// TIA Portal V20 export
FUNCTION "CALL_OPMODE_PANEL_FC" : Void   // FC200, LAD
TITLE = Aufruf Pult / Betriebsart / Call panels / operating modes
{ S7_Optimized_Access := 'TRUE' }
FAMILY : Base
VERSION : 1.0
// FUNKTIONSBESCHREIBUNG:
// Der Baustein dient als Aufrufschnittstelle für die HMI-/Panel- und Betriebsartenbausteine.
// Weitere Hinweise: siehe SICAR anwenderdefinierte Dokumentation / SICAR Online-Hilfe.
// DESCRIPTION OF FUNCTIONS:
// This function is the calling interface for initialization HMI/Panel and Operation mode blocks.
// For more informations see Tesla userdefined documentation / online-help.
// 描述 OF 功能:
// 这个 功能 is  calling 接口 给 初始化 HMI/Panel 和 运行 模式 blocks.
// 给 more informations see SICAR userdefined documentation / SICAR online-帮助.
// stored: AutoNumber false, SetENOAutomatically false
   VAR_TEMP
      Auxiliary_flag : Bool;
      Dummy_byte : Byte;
      dummy_word : Word;
      ParaAlarm : USInt;
      "020RB01_SlowDown" : Bool;
      "020RB02_SlowDown" : Bool;
      "020RB03_SlowDown" : Bool;
      "020RB04_SlowDown" : Bool;
      "020RB06_SlowDown" : Bool;
      "025RB01_SlowDown" : Bool;
      "025RB02_SlowDown" : Bool;
      "030RB01_SlowDown" : Bool;
      "030RB02_SlowDown" : Bool;
      "030RB03_SlowDown" : Bool;
      "030RB04_SlowDown" : Bool;
      待关联外部按钮1 : Bool;
      待关联外部按钮2 : Bool;
      待关联外部按钮2_1 : Bool;
   END_VAR
   VAR_TEMP   // added for the SCL form of the ladder/FBD networks
      _w1 : Bool;
      _w2 : Bool;
   END_VAR
BEGIN

REGION Network 1: Aufruf: HMI 1 / Call Operatorpanel_01: UBM1+010-HMI02 / Call: HMI_1
   // 介绍：设置和管理操作面板，
   // HMI:控制操作模式，可视化屏幕，
   // Panel：控制操作模式，按钮盒，
   // 有几个HMI调用几次，每次调用都需要对其定义类型。
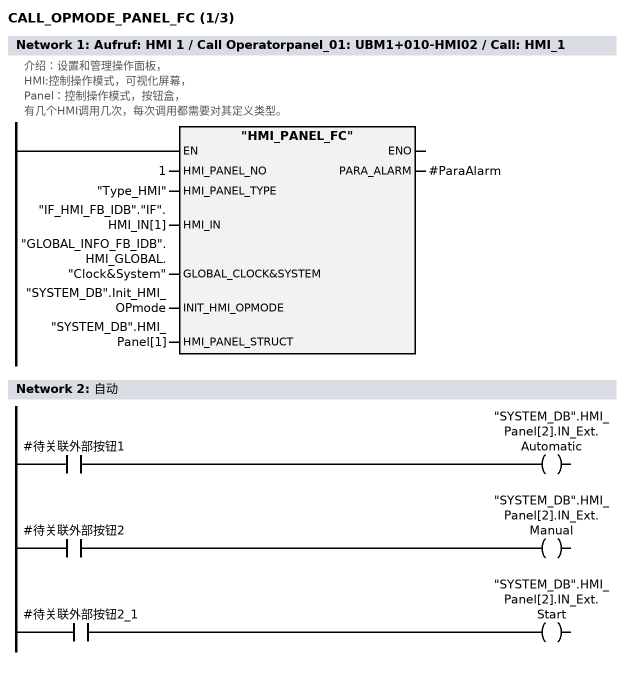
   RUNG wire#powerrail
      "HMI_PANEL_FC"(HMI_PANEL_NO := 1, HMI_PANEL_TYPE := "Type_HMI", HMI_IN := "IF_HMI_FB_IDB"."IF".HMI_IN[1], "GLOBAL_CLOCK&SYSTEM" := "GLOBAL_INFO_FB_IDB".HMI_GLOBAL."Clock&System", INIT_HMI_OPMODE := "SYSTEM_DB".Init_HMI_OPmode, HMI_PANEL_STRUCT := "SYSTEM_DB".HMI_Panel[1], PARA_ALARM => #ParaAlarm)
   END_RUNG
   // the same network as SCL:
   "HMI_PANEL_FC"(HMI_PANEL_NO := 1,
                  HMI_PANEL_TYPE := "Type_HMI",
                  HMI_IN := "IF_HMI_FB_IDB"."IF".HMI_IN[1],
                  "GLOBAL_CLOCK&SYSTEM" := "GLOBAL_INFO_FB_IDB".HMI_GLOBAL."Clock&System",
                  INIT_HMI_OPMODE := "SYSTEM_DB".Init_HMI_OPmode,
                  HMI_PANEL_STRUCT := "SYSTEM_DB".HMI_Panel[1],
                  PARA_ALARM => #ParaAlarm);
END_REGION

REGION Network 2: 自动
   RUNG wire#powerrail
      Contact( #待关联外部按钮1 )
      Coil( "SYSTEM_DB".HMI_Panel[2].IN_Ext.Automatic )
   END_RUNG
   RUNG wire#powerrail
      Contact( #待关联外部按钮2 )
      Coil( "SYSTEM_DB".HMI_Panel[2].IN_Ext.Manual )
   END_RUNG
   RUNG wire#powerrail
      Contact( #待关联外部按钮2_1 )
      Coil( "SYSTEM_DB".HMI_Panel[2].IN_Ext.Start )
   END_RUNG
   // the same network as SCL:
   "SYSTEM_DB".HMI_Panel[2].IN_Ext.Automatic := #待关联外部按钮1;
   "SYSTEM_DB".HMI_Panel[2].IN_Ext.Manual := #待关联外部按钮2;
   "SYSTEM_DB".HMI_Panel[2].IN_Ext.Start := #待关联外部按钮2_1;
END_REGION

REGION Network 3: E-Stop / Call: 运行 模式 area 1 - Create 新的 OpMode
   // 介绍：设置和管理操作操作模式OPMode，有几个OPMode就需要调用几次，每次调用都需要对其与HMI的关系进行定义。
   // 一个OPMode至少需要一个HMI/pannei控制；
   // 一个HMI/Panel可以控制多个OPMode；
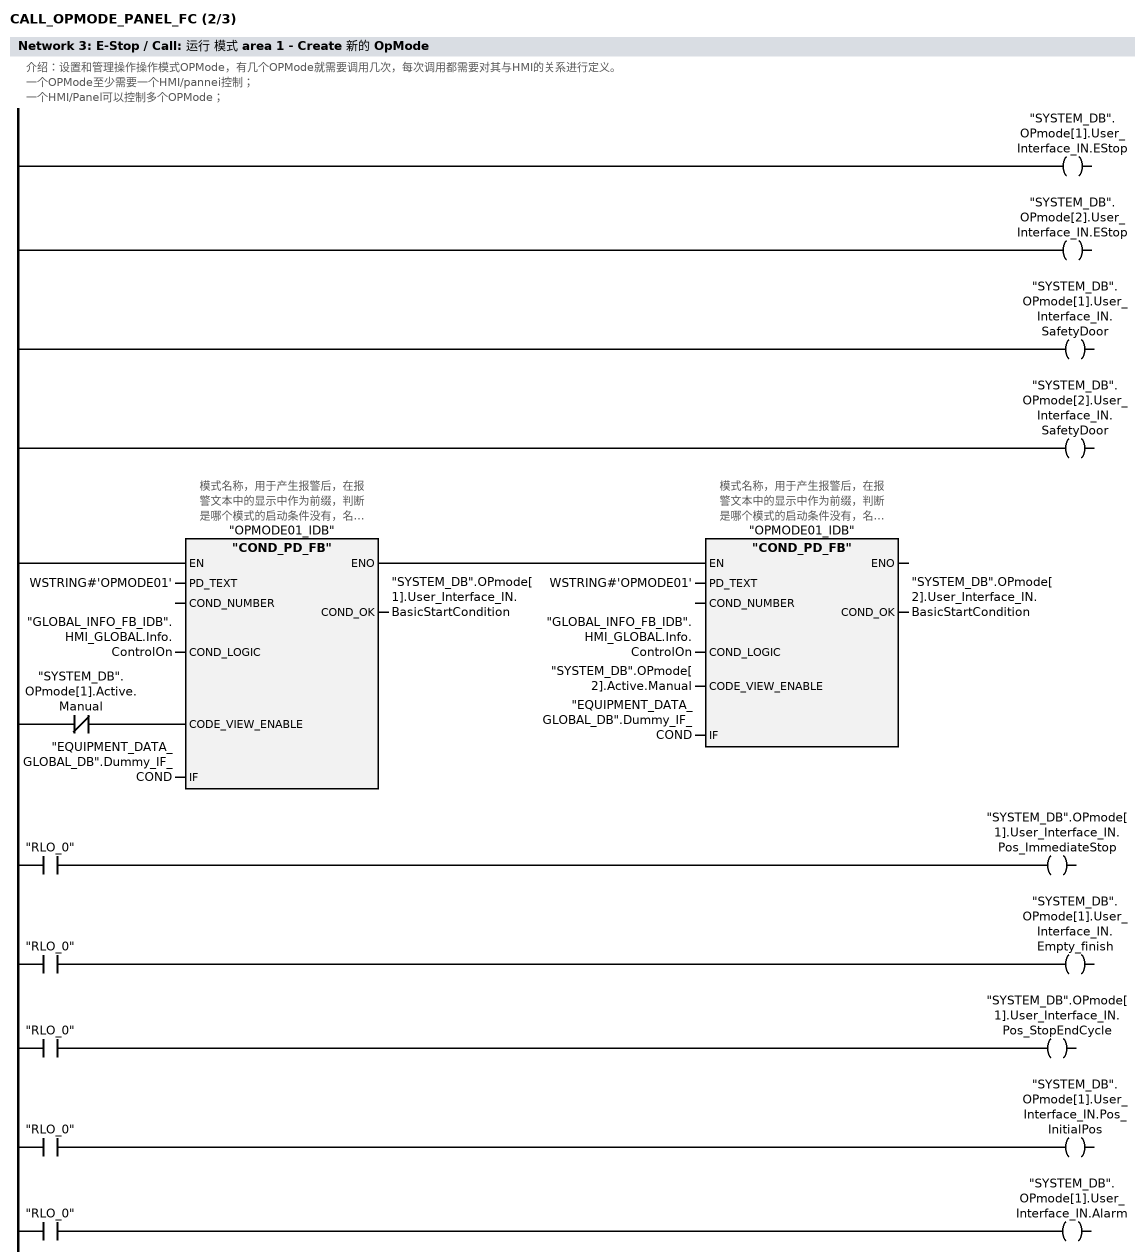
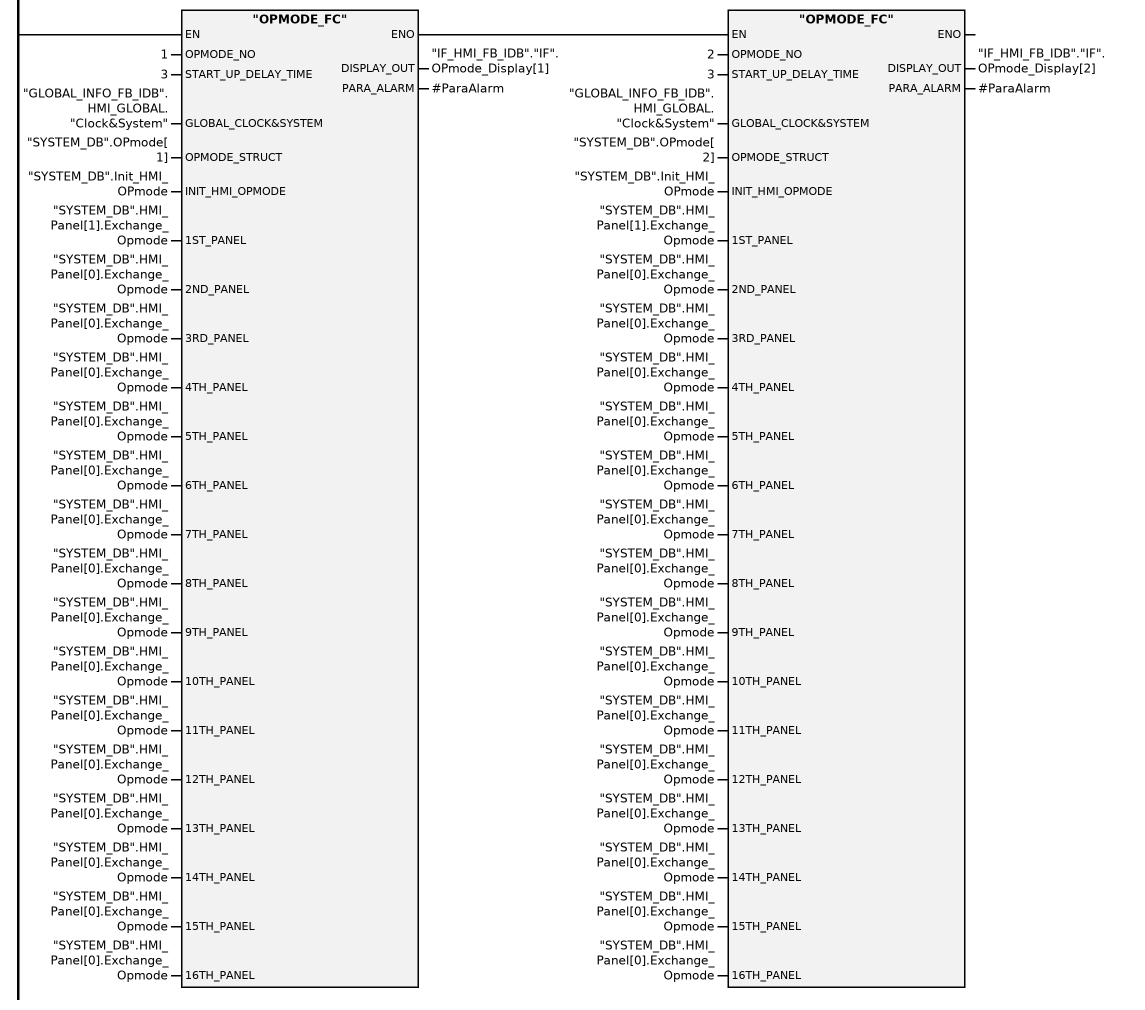
   RUNG wire#powerrail
      Coil( "SYSTEM_DB".OPmode[1].User_Interface_IN.EStop )
   END_RUNG
   RUNG wire#powerrail
      Coil( "SYSTEM_DB".OPmode[2].User_Interface_IN.EStop )
   END_RUNG
   RUNG wire#powerrail
      Coil( "SYSTEM_DB".OPmode[1].User_Interface_IN.SafetyDoor )
   END_RUNG
   RUNG wire#powerrail
      Coil( "SYSTEM_DB".OPmode[2].User_Interface_IN.SafetyDoor )
   END_RUNG
   RUNG wire#powerrail
      "OPMODE01_IDB"(CODE_VIEW_ENABLE := wire#w1, PD_TEXT := WSTRING#'OPMODE01', COND_NUMBER :=, COND_LOGIC := "GLOBAL_INFO_FB_IDB".HMI_GLOBAL.Info.ControlOn, "IF" := "EQUIPMENT_DATA_GLOBAL_DB".Dummy_IF_COND, COND_OK => "SYSTEM_DB".OPmode[1].User_Interface_IN.BasicStartCondition)   // 模式名称，用于产生报警后，在报警文本中的显示中作为前缀，判断是哪个模式的启动条件没有，名称已经预先填写在了对应DB块数据中
      "OPMODE01_IDB"(PD_TEXT := WSTRING#'OPMODE01', COND_NUMBER :=, COND_LOGIC := "GLOBAL_INFO_FB_IDB".HMI_GLOBAL.Info.ControlOn, CODE_VIEW_ENABLE := "SYSTEM_DB".OPmode[2].Active.Manual, "IF" := "EQUIPMENT_DATA_GLOBAL_DB".Dummy_IF_COND, COND_OK => "SYSTEM_DB".OPmode[2].User_Interface_IN.BasicStartCondition)   // 模式名称，用于产生报警后，在报警文本中的显示中作为前缀，判断是哪个模式的启动条件没有，名称已经预先填写在了对应DB块数据中
   END_RUNG
   RUNG wire#powerrail
      I_Contact( "SYSTEM_DB".OPmode[1].Active.Manual )
   END_RUNG wire#w1
   RUNG wire#powerrail
      Contact( "RLO_0" )
      Coil( "SYSTEM_DB".OPmode[1].User_Interface_IN.Pos_ImmediateStop )
   END_RUNG
   RUNG wire#powerrail
      Contact( "RLO_0" )
      Coil( "SYSTEM_DB".OPmode[1].User_Interface_IN.Empty_finish )
   END_RUNG
   RUNG wire#powerrail
      Contact( "RLO_0" )
      Coil( "SYSTEM_DB".OPmode[1].User_Interface_IN.Pos_StopEndCycle )
   END_RUNG
   RUNG wire#powerrail
      Contact( "RLO_0" )
      Coil( "SYSTEM_DB".OPmode[1].User_Interface_IN.Pos_InitialPos )
   END_RUNG
   RUNG wire#powerrail
      Contact( "RLO_0" )
      Coil( "SYSTEM_DB".OPmode[1].User_Interface_IN.Alarm )
   END_RUNG
   RUNG wire#powerrail
      "OPMODE_FC"(OPMODE_NO := 1, START_UP_DELAY_TIME := 3, "GLOBAL_CLOCK&SYSTEM" := "GLOBAL_INFO_FB_IDB".HMI_GLOBAL."Clock&System", OPMODE_STRUCT := "SYSTEM_DB".OPmode[1], INIT_HMI_OPMODE := "SYSTEM_DB".Init_HMI_OPmode, "1ST_PANEL" := "SYSTEM_DB".HMI_Panel[1].Exchange_Opmode, "2ND_PANEL" := "SYSTEM_DB".HMI_Panel[0].Exchange_Opmode, "3RD_PANEL" := "SYSTEM_DB".HMI_Panel[0].Exchange_Opmode, "4TH_PANEL" := "SYSTEM_DB".HMI_Panel[0].Exchange_Opmode, "5TH_PANEL" := "SYSTEM_DB".HMI_Panel[0].Exchange_Opmode, "6TH_PANEL" := "SYSTEM_DB".HMI_Panel[0].Exchange_Opmode, "7TH_PANEL" := "SYSTEM_DB".HMI_Panel[0].Exchange_Opmode, "8TH_PANEL" := "SYSTEM_DB".HMI_Panel[0].Exchange_Opmode, "9TH_PANEL" := "SYSTEM_DB".HMI_Panel[0].Exchange_Opmode, "10TH_PANEL" := "SYSTEM_DB".HMI_Panel[0].Exchange_Opmode, "11TH_PANEL" := "SYSTEM_DB".HMI_Panel[0].Exchange_Opmode, "12TH_PANEL" := "SYSTEM_DB".HMI_Panel[0].Exchange_Opmode, "13TH_PANEL" := "SYSTEM_DB".HMI_Panel[0].Exchange_Opmode, "14TH_PANEL" := "SYSTEM_DB".HMI_Panel[0].Exchange_Opmode, "15TH_PANEL" := "SYSTEM_DB".HMI_Panel[0].Exchange_Opmode, "16TH_PANEL" := "SYSTEM_DB".HMI_Panel[0].Exchange_Opmode, DISPLAY_OUT => "IF_HMI_FB_IDB"."IF".OPmode_Display[1], PARA_ALARM => #ParaAlarm)
      "OPMODE_FC"(OPMODE_NO := 2, START_UP_DELAY_TIME := 3, "GLOBAL_CLOCK&SYSTEM" := "GLOBAL_INFO_FB_IDB".HMI_GLOBAL."Clock&System", OPMODE_STRUCT := "SYSTEM_DB".OPmode[2], INIT_HMI_OPMODE := "SYSTEM_DB".Init_HMI_OPmode, "1ST_PANEL" := "SYSTEM_DB".HMI_Panel[1].Exchange_Opmode, "2ND_PANEL" := "SYSTEM_DB".HMI_Panel[0].Exchange_Opmode, "3RD_PANEL" := "SYSTEM_DB".HMI_Panel[0].Exchange_Opmode, "4TH_PANEL" := "SYSTEM_DB".HMI_Panel[0].Exchange_Opmode, "5TH_PANEL" := "SYSTEM_DB".HMI_Panel[0].Exchange_Opmode, "6TH_PANEL" := "SYSTEM_DB".HMI_Panel[0].Exchange_Opmode, "7TH_PANEL" := "SYSTEM_DB".HMI_Panel[0].Exchange_Opmode, "8TH_PANEL" := "SYSTEM_DB".HMI_Panel[0].Exchange_Opmode, "9TH_PANEL" := "SYSTEM_DB".HMI_Panel[0].Exchange_Opmode, "10TH_PANEL" := "SYSTEM_DB".HMI_Panel[0].Exchange_Opmode, "11TH_PANEL" := "SYSTEM_DB".HMI_Panel[0].Exchange_Opmode, "12TH_PANEL" := "SYSTEM_DB".HMI_Panel[0].Exchange_Opmode, "13TH_PANEL" := "SYSTEM_DB".HMI_Panel[0].Exchange_Opmode, "14TH_PANEL" := "SYSTEM_DB".HMI_Panel[0].Exchange_Opmode, "15TH_PANEL" := "SYSTEM_DB".HMI_Panel[0].Exchange_Opmode, "16TH_PANEL" := "SYSTEM_DB".HMI_Panel[0].Exchange_Opmode, DISPLAY_OUT => "IF_HMI_FB_IDB"."IF".OPmode_Display[2], PARA_ALARM => #ParaAlarm)
   END_RUNG
   // the same network as SCL:
   "SYSTEM_DB".OPmode[1].User_Interface_IN.EStop := TRUE;
   "SYSTEM_DB".OPmode[2].User_Interface_IN.EStop := TRUE;
   "SYSTEM_DB".OPmode[1].User_Interface_IN.SafetyDoor := TRUE;
   "SYSTEM_DB".OPmode[2].User_Interface_IN.SafetyDoor := TRUE;
   "OPMODE01_IDB"(PD_TEXT := WSTRING#'OPMODE01',   // "COND_PD_FB": 模式名称，用于产生报警后，在报警文本中的显示中作为前缀，判断是哪个模式的启动条件没有，名称已经预先填写在了对应DB块数据中
                  COND_LOGIC := "GLOBAL_INFO_FB_IDB".HMI_GLOBAL.Info.ControlOn,
                  CODE_VIEW_ENABLE := NOT "SYSTEM_DB".OPmode[1].Active.Manual,
                  "IF" := "EQUIPMENT_DATA_GLOBAL_DB".Dummy_IF_COND,
                  COND_OK => "SYSTEM_DB".OPmode[1].User_Interface_IN.BasicStartCondition,
                  ENO => #_w1);
   IF #_w1 THEN
       "OPMODE01_IDB"(PD_TEXT := WSTRING#'OPMODE01',   // "COND_PD_FB": 模式名称，用于产生报警后，在报警文本中的显示中作为前缀，判断是哪个模式的启动条件没有，名称已经预先填写在了对应DB块数据中
                      COND_LOGIC := "GLOBAL_INFO_FB_IDB".HMI_GLOBAL.Info.ControlOn,
                      CODE_VIEW_ENABLE := "SYSTEM_DB".OPmode[2].Active.Manual,
                      "IF" := "EQUIPMENT_DATA_GLOBAL_DB".Dummy_IF_COND,
                      COND_OK => "SYSTEM_DB".OPmode[2].User_Interface_IN.BasicStartCondition);
   END_IF;
   "SYSTEM_DB".OPmode[1].User_Interface_IN.Pos_ImmediateStop := "RLO_0";
   "SYSTEM_DB".OPmode[1].User_Interface_IN.Empty_finish := "RLO_0";
   "SYSTEM_DB".OPmode[1].User_Interface_IN.Pos_StopEndCycle := "RLO_0";
   "SYSTEM_DB".OPmode[1].User_Interface_IN.Pos_InitialPos := "RLO_0";
   "SYSTEM_DB".OPmode[1].User_Interface_IN.Alarm := "RLO_0";
   "OPMODE_FC"(OPMODE_NO := 1,
               START_UP_DELAY_TIME := 3,
               "GLOBAL_CLOCK&SYSTEM" := "GLOBAL_INFO_FB_IDB".HMI_GLOBAL."Clock&System",
               OPMODE_STRUCT := "SYSTEM_DB".OPmode[1],
               INIT_HMI_OPMODE := "SYSTEM_DB".Init_HMI_OPmode,
               "1ST_PANEL" := "SYSTEM_DB".HMI_Panel[1].Exchange_Opmode,
               "2ND_PANEL" := "SYSTEM_DB".HMI_Panel[0].Exchange_Opmode,
               "3RD_PANEL" := "SYSTEM_DB".HMI_Panel[0].Exchange_Opmode,
               "4TH_PANEL" := "SYSTEM_DB".HMI_Panel[0].Exchange_Opmode,
               "5TH_PANEL" := "SYSTEM_DB".HMI_Panel[0].Exchange_Opmode,
               "6TH_PANEL" := "SYSTEM_DB".HMI_Panel[0].Exchange_Opmode,
               "7TH_PANEL" := "SYSTEM_DB".HMI_Panel[0].Exchange_Opmode,
               "8TH_PANEL" := "SYSTEM_DB".HMI_Panel[0].Exchange_Opmode,
               "9TH_PANEL" := "SYSTEM_DB".HMI_Panel[0].Exchange_Opmode,
               "10TH_PANEL" := "SYSTEM_DB".HMI_Panel[0].Exchange_Opmode,
               "11TH_PANEL" := "SYSTEM_DB".HMI_Panel[0].Exchange_Opmode,
               "12TH_PANEL" := "SYSTEM_DB".HMI_Panel[0].Exchange_Opmode,
               "13TH_PANEL" := "SYSTEM_DB".HMI_Panel[0].Exchange_Opmode,
               "14TH_PANEL" := "SYSTEM_DB".HMI_Panel[0].Exchange_Opmode,
               "15TH_PANEL" := "SYSTEM_DB".HMI_Panel[0].Exchange_Opmode,
               "16TH_PANEL" := "SYSTEM_DB".HMI_Panel[0].Exchange_Opmode,
               DISPLAY_OUT => "IF_HMI_FB_IDB"."IF".OPmode_Display[1],
               PARA_ALARM => #ParaAlarm,
               ENO => #_w2);
   IF #_w2 THEN
       "OPMODE_FC"(OPMODE_NO := 2,
                   START_UP_DELAY_TIME := 3,
                   "GLOBAL_CLOCK&SYSTEM" := "GLOBAL_INFO_FB_IDB".HMI_GLOBAL."Clock&System",
                   OPMODE_STRUCT := "SYSTEM_DB".OPmode[2],
                   INIT_HMI_OPMODE := "SYSTEM_DB".Init_HMI_OPmode,
                   "1ST_PANEL" := "SYSTEM_DB".HMI_Panel[1].Exchange_Opmode,
                   "2ND_PANEL" := "SYSTEM_DB".HMI_Panel[0].Exchange_Opmode,
                   "3RD_PANEL" := "SYSTEM_DB".HMI_Panel[0].Exchange_Opmode,
                   "4TH_PANEL" := "SYSTEM_DB".HMI_Panel[0].Exchange_Opmode,
                   "5TH_PANEL" := "SYSTEM_DB".HMI_Panel[0].Exchange_Opmode,
                   "6TH_PANEL" := "SYSTEM_DB".HMI_Panel[0].Exchange_Opmode,
                   "7TH_PANEL" := "SYSTEM_DB".HMI_Panel[0].Exchange_Opmode,
                   "8TH_PANEL" := "SYSTEM_DB".HMI_Panel[0].Exchange_Opmode,
                   "9TH_PANEL" := "SYSTEM_DB".HMI_Panel[0].Exchange_Opmode,
                   "10TH_PANEL" := "SYSTEM_DB".HMI_Panel[0].Exchange_Opmode,
                   "11TH_PANEL" := "SYSTEM_DB".HMI_Panel[0].Exchange_Opmode,
                   "12TH_PANEL" := "SYSTEM_DB".HMI_Panel[0].Exchange_Opmode,
                   "13TH_PANEL" := "SYSTEM_DB".HMI_Panel[0].Exchange_Opmode,
                   "14TH_PANEL" := "SYSTEM_DB".HMI_Panel[0].Exchange_Opmode,
                   "15TH_PANEL" := "SYSTEM_DB".HMI_Panel[0].Exchange_Opmode,
                   "16TH_PANEL" := "SYSTEM_DB".HMI_Panel[0].Exchange_Opmode,
                   DISPLAY_OUT => "IF_HMI_FB_IDB"."IF".OPmode_Display[2],
                   PARA_ALARM => #ParaAlarm);
   END_IF;
END_REGION

REGION Network 4: Aufruf: HMI Schnittstelle / Call HMI_IF_FB
   // 介绍：HMI与PLC系统的接口功能块，
   // 此块用来管理所有的HMIheOPMode操作模式的接口，用户不需要对此做任何修改。
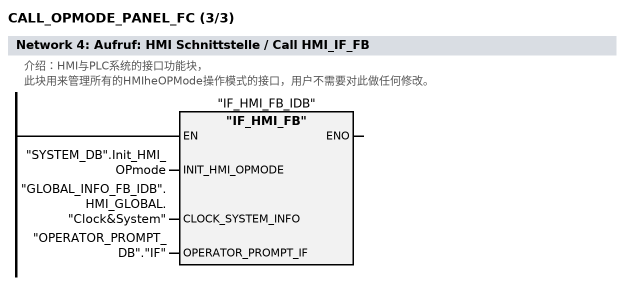
   RUNG wire#powerrail
      "IF_HMI_FB_IDB"(INIT_HMI_OPMODE := "SYSTEM_DB".Init_HMI_OPmode, CLOCK_SYSTEM_INFO := "GLOBAL_INFO_FB_IDB".HMI_GLOBAL."Clock&System", OPERATOR_PROMPT_IF := "OPERATOR_PROMPT_DB"."IF")
   END_RUNG
   // the same network as SCL:
   "IF_HMI_FB_IDB"(INIT_HMI_OPMODE := "SYSTEM_DB".Init_HMI_OPmode,   // "IF_HMI_FB"
                   CLOCK_SYSTEM_INFO := "GLOBAL_INFO_FB_IDB".HMI_GLOBAL."Clock&System",
                   OPERATOR_PROMPT_IF := "OPERATOR_PROMPT_DB"."IF");
END_REGION
END_FUNCTION
